TYPE Mes1 :
STRUCT
	rExcelRate	:ARRAY[0..119] OF REAL;	//优报表real
	uOther		:ARRAY[0..19] OF UINT;	//信号交互
	bFuncEN      :ARRAY[0..50] OF BOOL;  //功能开关状态
	Error       :ARRAY[0..50] OF BOOL;  //功能开关状态报警
END_STRUCT
END_TYPE

(* stored: Version 1.1.0.1, ProductVersion 3.1.4024.12
   DUT Mes1: Id {1340bf3e-7d1a-4d42-b2c8-b196f1c74404} *)
